FUNCTION_BLOCK T_ProductionToMaintenaceInAbort EXTENDS T_UnitTestBase
VAR
  em : EquipmentModule; 
  actual, expected : E_PMLUnitMode;
	scanCounter: INT;

  myTestState : (ARRANGE,CMD, ACT, ASSERT);
END_VAR

CASE myTestState OF
  ARRANGE:
    em.CyclicLogic();

    IF em.InitComplete THEN
      myTestState := CMD;
    END_IF

  CMD:
    em.ChangeMode(E_PMLUnitMode.ePMLUnitMode_Maintenance);
    myTestState := ACT;
    
  ACT:
    em.CyclicLogic();
    
    IF CycleModuleLogicToAllowChangesToFilterThrough() THEN
      actual := em.CurrentMode;
      expected := E_PMLUnitMode.ePMLUnitMode_Maintenance;
      myTestState := ASSERT;
    END_IF

  ASSERT:
    assertion.AssertEquals_UINT(TO_UINT(actual), TO_UINT(expected), 'actual := equipmentModule.CurrentMode');
END_CASE

METHOD CycleModuleLogicToAllowChangesToFilterThrough : BOOL
VAR_INST
	i: INT;

END_VAR
em.CyclicLogic();
CycleModuleLogicToAllowChangesToFilterThrough := i >= 10;
i := SEL(i >= 10, i + 1, 0);
END_METHOD

END_FUNCTION_BLOCK

(* stored: Version 1.1.0.1, ProductVersion 3.1.4024.12
   POU T_ProductionToMaintenaceInAbort: Id {543f2245-bb84-43df-8d57-c030fa48510c}, SpecialFunc None
   Method CycleModuleLogicToAllowChangesToFilterThrough: Id {ce1e0657-9a35-4670-a8f1-a85b709101bb} *)
